SUBAPPLICATION Button_IXA_TO_logiBUS_QXA_BG_OPC_LATCHING (* Button IXA -> logiBUS QXA + Hintergrundfarbe, plus OPC-UA Read/Write (generisch, ein Kanal) - Klick-Toggle-Variante (SR-Latch) *)
  (* Standard: 61499-2; Description: Copyright (c) 2023 Meisterschulen am Ostbahnhof This program and the accompanying materials are made available under the terms of the Eclipse Public License 2.0 which is available at https://www.eclipse.org/legal/epl-2.0/ SPDX-License-Identifier: EPL-2.0 *)
  (* Version 1.1, 2026-07-20, Franz Höpfinger, Meisterschulen am Ostbahnhof, Background *)
  (* Version 1.0, 2026-01-15, Franz Höpfinger, Meisterschulen am Ostbahnhof, initial API and implementation and/or initial documentation *)
  PACKAGE MyLib::sys;
  IMPORT isobus::UT::Q::const::IDs::ID_NULL;
  IMPORT logiBUS::io::DQ::logiBUS_DO;
  IMPORT logiBUS::io::DQ::logiBUS_DO_S;
  (* Documentation:
  Button → logiBUS-Ausgang mit Klick-Toggle (SR-Latch)
   Latching-Variante von Button_IXA_TO_logiBUS_QXA_BG_OPC: lokaler VT-Button UND Remote-OPC-UA-Kommando werden je über AX_ASR_RF_TRIG in Set/Reset-Events gewandelt, per ASR_MERGE_2 zusammengeführt und in ASR_AX_SR gelatcht (Last-Wins) - ein Klick schaltet den Ausgang EIN, ein zweiter Klick AUS, unabhängig davon wie lange gedrückt wird.
   Aufbewahrt für den Fall, dass das Klick-Toggle-Verhalten wieder gebraucht wird - seit 2026-09-07 verwendet Button_IXA_TO_logiBUS_QXA_BG_OPC selbst stattdessen ein einfaches AX_OR_2 (tastend/momentary, kein Latch). Gleiches Interface (u16ObjId/Output/ID_READ/ID_WRITE), 1:1 austauschbar.
  *)
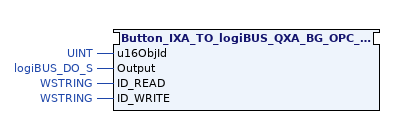
  VAR_INPUT
    u16ObjId : UINT := ID_NULL; (* Object ID Button/Hintergrund (VT), ID_NULL = noch kein VT-Objekt *)
    Output : logiBUS::io::DQ::logiBUS_DO_S := logiBUS_DO::Invalid; (* Identify the Output Output_Q1..Q12 *)
    ID_READ : WSTRING; (* OPC-UA Subscribe-Key (schreibbar) *)
    ID_WRITE : WSTRING; (* OPC-UA Publish-Key (lesbar) *)
  END_VAR
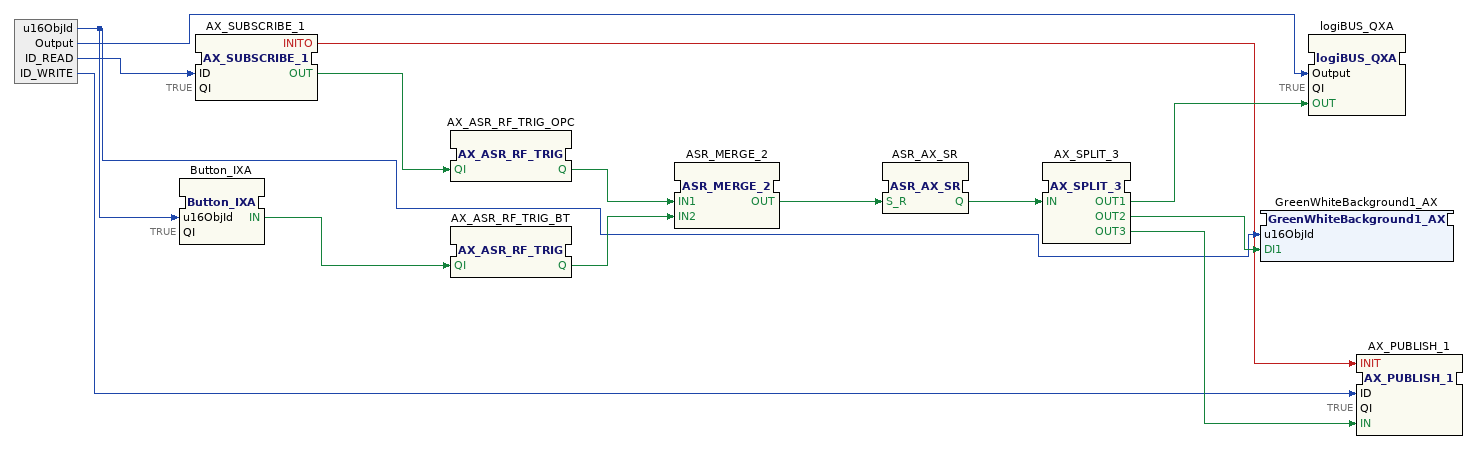
  FBS
    logiBUS_QXA : logiBUS::io::DQ::logiBUS_QXA(QI := TRUE);
    Button_IXA : isobus::UT::io::Button::Button_IXA(QI := TRUE);
    AX_SPLIT_3 : adapter::events::unidirectional::AX_SPLIT_3;
    AX_SUBSCRIBE_1 : adapter::net::AX_SUBSCRIBE_1(QI := TRUE);
    AX_PUBLISH_1 : adapter::net::AX_PUBLISH_1(QI := TRUE);
    AX_ASR_RF_TRIG_BT : adapter::events::unidirectional::AX_ASR_RF_TRIG;
    ASR_AX_SR : adapter::events::unidirectional::ASR_AX_SR;
    AX_ASR_RF_TRIG_OPC : adapter::events::unidirectional::AX_ASR_RF_TRIG;
    ASR_MERGE_2 : adapter::events::unidirectional::ASR_MERGE_2;
  END_FBS
  SUBAPPS
    GreenWhiteBackground1_AX : MyLib::sys::GreenWhiteBackground1_AX;
  END_SUBAPPS
  EVENT_CONNECTIONS
    AX_SUBSCRIBE_1.INITO TO AX_PUBLISH_1.INIT;
  END_CONNECTIONS
  DATA_CONNECTIONS
    u16ObjId TO Button_IXA.u16ObjId;
    Output TO logiBUS_QXA.Output;
    u16ObjId TO GreenWhiteBackground1_AX.u16ObjId;
    ID_READ TO AX_SUBSCRIBE_1.ID;
    ID_WRITE TO AX_PUBLISH_1.ID;
  END_CONNECTIONS
  ADAPTER_CONNECTIONS
    Button_IXA.IN TO AX_ASR_RF_TRIG_BT.QI;
    AX_SPLIT_3.OUT1 TO logiBUS_QXA.OUT;
    AX_SPLIT_3.OUT2 TO GreenWhiteBackground1_AX.DI1;
    ASR_AX_SR.Q TO AX_SPLIT_3.IN;
    AX_SUBSCRIBE_1.OUT TO AX_ASR_RF_TRIG_OPC.QI;
    AX_SPLIT_3.OUT3 TO AX_PUBLISH_1.IN;
    AX_ASR_RF_TRIG_OPC.Q TO ASR_MERGE_2.IN1;
    AX_ASR_RF_TRIG_BT.Q TO ASR_MERGE_2.IN2;
    ASR_MERGE_2.OUT TO ASR_AX_SR.S_R;
  END_CONNECTIONS
END_SUBAPPLICATION
